INTERFACE ITF_BaseDescriptor

METHOD PUBLIC GetDefaultValue : REAL
VAR_INPUT
END_VAR
END_METHOD

METHOD PUBLIC GetMax : REAL
VAR_INPUT
END_VAR
END_METHOD

METHOD PUBLIC GetMin : REAL
VAR_INPUT
END_VAR
END_METHOD

METHOD PUBLIC GetTexts : ST_BaseLabel
VAR_INPUT
END_VAR
END_METHOD

METHOD PUBLIC GetUnit : STRING(6)
VAR_INPUT
END_VAR
END_METHOD

METHOD PUBLIC GetValue : REAL
VAR_INPUT
END_VAR
END_METHOD

METHOD PUBLIC SetDefaultValue
VAR_INPUT
	rDefaultValue: REAL;
END_VAR
END_METHOD

METHOD PUBLIC SetMax
VAR_INPUT
	rMax: REAL;
END_VAR
END_METHOD

METHOD PUBLIC SetMin
VAR_INPUT
	rMin: REAL;
END_VAR
END_METHOD

METHOD PUBLIC SetText
VAR_INPUT
	eLocation			: E_BaseLocation;
	wsDescription		: WSTRING;
END_VAR
END_METHOD

METHOD PUBLIC SetTexts
VAR_INPUT
	stTexts				: ST_BaseLabel;
END_VAR
END_METHOD

METHOD PUBLIC SetUnit
VAR_INPUT
	sUnit: STRING(6);
END_VAR
END_METHOD

METHOD PUBLIC SetValue
VAR_INPUT
	rValue: REAL;
END_VAR
END_METHOD

END_INTERFACE

(* stored: Version 1.1.0.1
   Itf ITF_BaseDescriptor: Id {ada92c2f-1741-06d9-3083-5dca405ada51}
   Method GetDefaultValue: Id {0001106c-cdff-0475-27f0-eb00a18be38e}
   Method GetMax: Id {bae076a0-3150-01b8-3c53-4367e86f3b43}
   Method GetMin: Id {e657ef90-b27c-03de-0c7c-5543479dfc1c}
   Method GetTexts: Id {d80bba81-9353-01a2-25e9-143430746f38}
   Method GetUnit: Id {e28259f1-3474-03b8-0931-d0fb54d804c7}
   Method GetValue: Id {527925d6-48f4-0a8c-3620-625e15c2c437}
   Method SetDefaultValue: Id {b1fdf0f6-b449-078c-0cd0-63fd394ce2b9}
   Method SetMax: Id {224191b0-b2d2-0604-27db-6f5018206d35}
   Method SetMin: Id {636d9330-761a-01b1-09e9-9bea1c1f04aa}
   Method SetText: Id {a325a82c-37c7-0885-1304-9e7776739f28}
   Method SetTexts: Id {ac0a0a67-d616-01b6-2ae1-e67d6995b8d6}
   Method SetUnit: Id {063eb5d1-150b-042b-3b06-66430baeec81}
   Method SetValue: Id {28cee76f-1074-00e9-37db-eacf1b2c2368} *)
